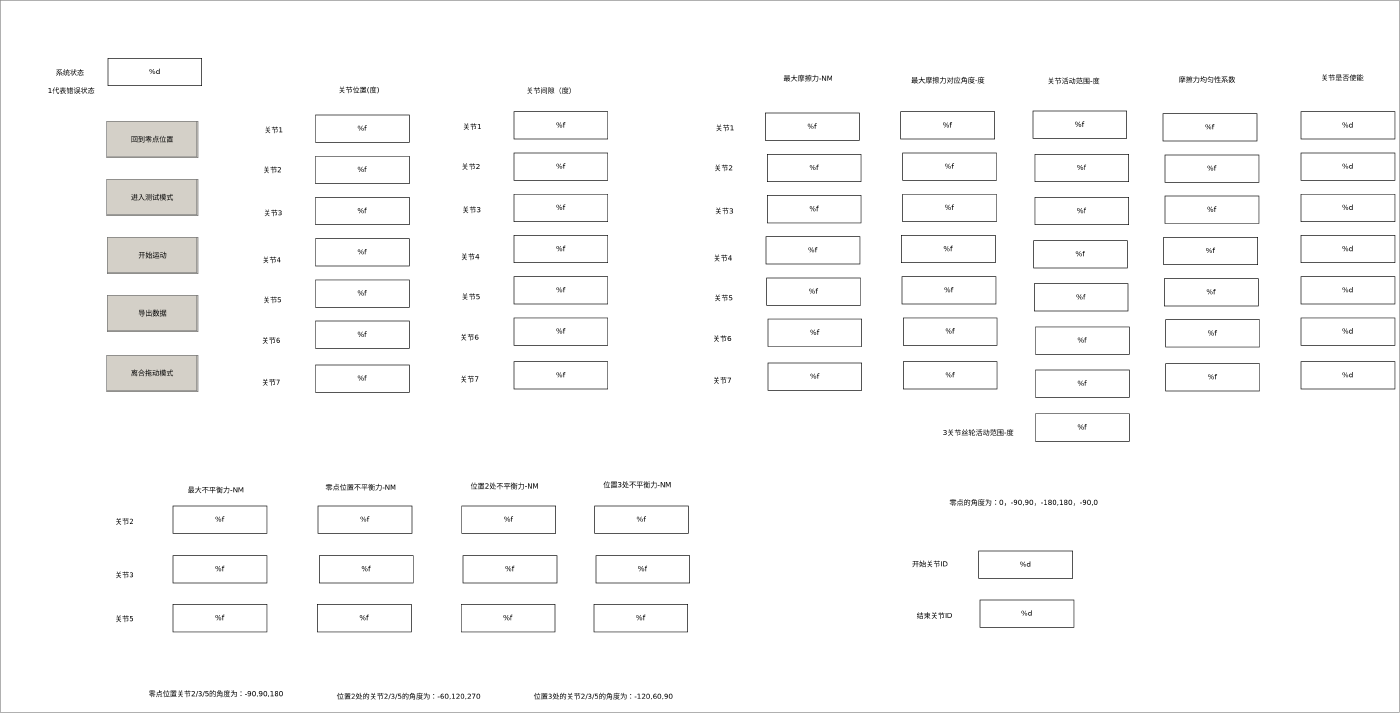
VISUALIZATION friction_a1  // 2172x1107
    Button (165,278 142x57), "进入测试模式", colour toggle: g_frictionTest.m_testMode[1]
        toggle g_frictionTest.m_testMode[1]
    Button (166,368 141x57), "开始运动", colour toggle: g_frictionTest.m_startMotion[1]
        toggle g_frictionTest.m_startMotion[1]
    Rectangle (489,178 146x43), "%f", text variable: g_frictionTest.m_armDHJntPos[1][1]
    Label (373,184 103x36), "关节1"
    Label (371,246 103x36), "关节2"
    Label (372,313 103x36), "关节3"
    Label (370,386 103x36), "关节4"
    Label (371,448 103x36), "关节5"
    Label (369,511 103x36), "关节6"
    Label (369,576 103x36), "关节7"
    Rectangle (489,242 146x43), "%f", text variable: g_frictionTest.m_armDHJntPos[1][2]
    Rectangle (489,306 146x43), "%f", text variable: g_frictionTest.m_armDHJntPos[1][3]
    Rectangle (489,370 146x43), "%f", text variable: g_frictionTest.m_armDHJntPos[1][4]
    Rectangle (489,434 146x43), "%f", text variable: g_frictionTest.m_armDHJntPos[1][5]
    Rectangle (489,498 146x43), "%f", text variable: g_frictionTest.m_armDHJntPos[1][6]
    Rectangle (489,566 146x43), "%f", text variable: g_frictionTest.m_armDHJntPos[1][7]
    Button (165,551 142x57), "离合拖动模式", colour toggle: g_frictionTest.m_clutchMode[1]
        toggle g_frictionTest.m_clutchMode[1]
    Rectangle (797,173 146x43), "%f", text variable: g_frictionTest.m_jntGap[1][1]
    Label (681,179 103x36), "关节1"
    Label (679,241 103x36), "关节2"
    Label (680,308 103x36), "关节3"
    Label (678,381 103x36), "关节4"
    Label (679,443 103x36), "关节5"
    Label (677,506 103x36), "关节6"
    Label (677,571 103x36), "关节7"
    Rectangle (797,237 146x43), "%f", text variable: g_frictionTest.m_jntGap[1][2]
    Rectangle (797,301 146x43), "%f", text variable: g_frictionTest.m_jntGap[1][3]
    Rectangle (797,365 146x43), "%f", text variable: g_frictionTest.m_jntGap[1][4]
    Rectangle (797,429 146x43), "%f", text variable: g_frictionTest.m_jntGap[1][5]
    Rectangle (797,493 146x43), "%f", text variable: g_frictionTest.m_jntGap[1][6]
    Rectangle (797,561 146x43), "%f", text variable: g_frictionTest.m_jntGap[1][7]
    Label (118,795 150x30), "关节2"
    Label (118,878 150x30), "关节3"
    Label (118,946 150x30), "关节5"
    Rectangle (268,785 146x43), "%f", text variable: g_frictionTest.m_unbalancedMax[1][2]
    Rectangle (268,862 146x43), "%f", text variable: g_frictionTest.m_unbalancedMax[1][3]
    Rectangle (268,938 146x43), "%f", text variable: g_frictionTest.m_unbalancedMax[1][5]
    Rectangle (493,785 146x43), "%f", text variable: g_frictionTest.m_jntTestPntUnbalancedTrq[1,2,1]
    Rectangle (495,862 146x43), "%f", text variable: g_frictionTest.m_jntTestPntUnbalancedTrq[1,3,1]
    Rectangle (492,938 146x43), "%f", text variable: g_frictionTest.m_jntTestPntUnbalancedTrq[1,5,1]
    Rectangle (716,785 146x43), "%f", text variable: g_frictionTest.m_jntTestPntUnbalancedTrq[1,2,2]
    Rectangle (718,862 146x43), "%f", text variable: g_frictionTest.m_jntTestPntUnbalancedTrq[1,3,2]
    Rectangle (715,938 146x43), "%f", text variable: g_frictionTest.m_jntTestPntUnbalancedTrq[1,5,2]
    Rectangle (922,785 146x43), "%f", text variable: g_frictionTest.m_jntTestPntUnbalancedTrq[1,2,3]
    Rectangle (924,862 146x43), "%f", text variable: g_frictionTest.m_jntTestPntUnbalancedTrq[1,3,3]
    Rectangle (921,938 146x43), "%f", text variable: g_frictionTest.m_jntTestPntUnbalancedTrq[1,5,3]
    Button (166,458 141x57), "导出数据", colour toggle: g_frictionTest.m_duringWriteData[1]
        tap g_frictionTest.m_writeData[1]
    Label (184,1052 302x51), "零点位置关节2/3/5的角度为：-90,90,180"
    Label (483,1056 302x51), "位置2处的关节2/3/5的角度为：-60,120,270"
    Label (785,1056 302x51), "位置3处的关节2/3/5的角度为：-120,60,90"
    Label (260,746 150x30), "最大不平衡力-NM"
    Label (485,742 150x30), "零点位置不平衡力-NM"
    Label (708,740 150x30), "位置2处不平衡力-NM"
    Label (914,738 150x30), "位置3处不平衡力-NM"
    Label (1401,757 375x47), "零点的角度为：0，-90,90，-180,180，-90,0"
    Label (1368,861 150x30), "开始关节ID"
    Rectangle (1518,855 146x43), "%d", text variable: g_frictionTest.m_jntIdStart[1]
        OnMouseClick: write the text variable via Default
    Label (1375,941 150x30), "结束关节ID"
    Rectangle (1520,931 146x43), "%d", text variable: g_frictionTest.m_jntIdEnd[1]
        OnMouseClick: write the text variable via Default
    Label (482,125 150x30), "关节位置(度)"
    Label (780,126 150x30), "关节间隙（度）"
    Rectangle (1187,175 146x43), "%f", text variable: g_frictionTest.m_CoulombFrictionMax[1][1]
    Label (1073,181 103x36), "关节1"
    Label (1071,243 103x36), "关节2"
    Label (1072,310 103x36), "关节3"
    Label (1070,383 103x36), "关节4"
    Label (1071,445 103x36), "关节5"
    Label (1069,508 103x36), "关节6"
    Label (1069,573 103x36), "关节7"
    Rectangle (1190,239 146x43), "%f", text variable: g_frictionTest.m_CoulombFrictionMax[1][2]
    Rectangle (1190,303 146x43), "%f", text variable: g_frictionTest.m_CoulombFrictionMax[1][3]
    Rectangle (1188,367 146x43), "%f", text variable: g_frictionTest.m_CoulombFrictionMax[1][4]
    Rectangle (1189,431 146x43), "%f", text variable: g_frictionTest.m_CoulombFrictionMax[1][5]
    Rectangle (1191,495 146x43), "%f", text variable: g_frictionTest.m_CoulombFrictionMax[1][6]
    Rectangle (1191,563 146x43), "%f", text variable: g_frictionTest.m_CoulombFrictionMax[1][7]
    Label (1179,107 150x30), "最大摩擦力-NM"
    Rectangle (1397,173 146x43), "%f", text variable: g_frictionTest.m_CoulombFrictionMax_JntPos[1][1]
    Rectangle (1400,237 146x43), "%f", text variable: g_frictionTest.m_CoulombFrictionMax_JntPos[1][2]
    Rectangle (1400,301 146x43), "%f", text variable: g_frictionTest.m_CoulombFrictionMax_JntPos[1][3]
    Rectangle (1398,365 146x43), "%f", text variable: g_frictionTest.m_CoulombFrictionMax_JntPos[1][4]
    Rectangle (1399,429 146x43), "%f", text variable: g_frictionTest.m_CoulombFrictionMax_JntPos[1][5]
    Rectangle (1401,493 146x43), "%f", text variable: g_frictionTest.m_CoulombFrictionMax_JntPos[1][6]
    Rectangle (1401,561 146x43), "%f", text variable: g_frictionTest.m_CoulombFrictionMax_JntPos[1][7]
    Label (1354,110 233x30), "最大摩擦力对应角度-度"
    Rectangle (1602,172 146x43), "%f", text variable: g_frictionTest.m_jntMotRange[1][1]
    Rectangle (1605,239 146x43), "%f", text variable: g_frictionTest.m_jntMotRange[1][2]
    Rectangle (1605,306 146x43), "%f", text variable: g_frictionTest.m_jntMotRange[1][3]
    Rectangle (1603,373 146x43), "%f", text variable: g_frictionTest.m_jntMotRange[1][4]
    Rectangle (1604,440 146x43), "%f", text variable: g_frictionTest.m_jntMotRange[1][5]
    Rectangle (1606,507 146x43), "%f", text variable: g_frictionTest.m_jntMotRange[1][6]
    Rectangle (1606,574 146x43), "%f", text variable: g_frictionTest.m_jntMotRange[1][7]
    Label (1576,111 179x30), "关节活动范围-度"
    Button (165,188 142x57), "回到零点位置", colour toggle: g_frictionTest.m_getHome[1]
        tap g_frictionTest.m_getHome[1]
    Rectangle (167,90 146x43), "%d", text variable: g_systemInfo.m_masterArmState[1]
    Label (57,95 103x36), "系统状态"
    Label (59,123 103x36), "1代表错误状态"
    Rectangle (1606,642 146x43), "%f", text variable: g_frictionTest.m_jntMotRangeJ3[1]
    Label (1452,657 131x30), "3关节丝轮活动范围-度"
    Rectangle (1804,176 146x43), "%f", text variable: g_frictionTest.m_CoulombFrictionRatio[1,1]
    Rectangle (1807,240 146x43), "%f", text variable: g_frictionTest.m_CoulombFrictionRatio[1,2]
    Rectangle (1807,304 146x43), "%f", text variable: g_frictionTest.m_CoulombFrictionRatio[1,3]
    Rectangle (1805,368 146x43), "%f", text variable: g_frictionTest.m_CoulombFrictionRatio[1,4]
    Rectangle (1806,432 146x43), "%f", text variable: g_frictionTest.m_CoulombFrictionRatio[1,5]
    Rectangle (1808,496 146x43), "%f", text variable: g_frictionTest.m_CoulombFrictionRatio[1,6]
    Rectangle (1808,564 146x43), "%f", text variable: g_frictionTest.m_CoulombFrictionRatio[1,7]
    Label (1783,109 179x30), "摩擦力均匀性系数"
    Rectangle (2018,173 146x43), "%d", text variable: g_frictionTest.m_jntEnable[1,1]
        OnMouseClick: write the text variable via Default
    Label (1993,106 179x30), "关节是否使能"
    Rectangle (2018,237 146x43), "%d", text variable: g_frictionTest.m_jntEnable[1,2]
        OnMouseClick: write the text variable via Default
    Rectangle (2018,301 146x43), "%d", text variable: g_frictionTest.m_jntEnable[1,3]
        OnMouseClick: write the text variable via Default
    Rectangle (2018,365 146x43), "%d", text variable: g_frictionTest.m_jntEnable[1,4]
        OnMouseClick: write the text variable via Default
    Rectangle (2018,429 146x43), "%d", text variable: g_frictionTest.m_jntEnable[1,5]
        OnMouseClick: write the text variable via Default
    Rectangle (2018,493 146x43), "%d", text variable: g_frictionTest.m_jntEnable[1,6]
        OnMouseClick: write the text variable via Default
    Rectangle (2018,561 146x43), "%d", text variable: g_frictionTest.m_jntEnable[1,7]
        OnMouseClick: write the text variable via Default
END_VISUALIZATION

(* stored: Version 1.1.0.1, ProductVersion 3.1.4024.11
   Visu friction_a1: Id {831c13d7-b138-4dce-bd94-5dfa665395e3} *)
